FUNCTION_BLOCK F_REAL_TO_BOOL (* Service Interface Function Block Type *)
  (* Standard: 61131-3; Classification: standard type conversion function; Description: Copyright (c) 2013 Profactor GmbH This program and the accompanying materials are made available under the terms of the Eclipse Public License 2.0 which is available at https://www.eclipse.org/legal/epl-2.0/ SPDX-License-Identifier: EPL-2.0 *)
  (* Version 1.0, 2013-04-15, Matthias Plasch, Profactor GmbH *)
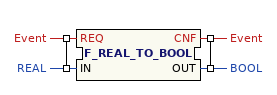
  EVENT_INPUT
    REQ WITH IN; (* Service Request *)
  END_EVENT
  EVENT_OUTPUT
    CNF WITH OUT; (* Confirmation of Requested Service *)
  END_EVENT
  VAR_INPUT
    IN : REAL; (* input value *)
  END_VAR
  VAR_OUTPUT
    OUT : BOOL; (* output value *)
  END_VAR
  (* Service APPLICATION/RESOURCE: Service Interface Function Block Type *)
END_FUNCTION_BLOCK
